FUNCTION_BLOCK FB_Test1000
VAR_INPUT
END_VAR
VAR_OUTPUT
END_VAR
VAR
	fbEvent: 			Tc3_Event.FB_Event;
	bVerbose:			BOOL;
	bInfo:				BOOL;
	bWarning:			BOOL;
	bError:				BOOL;
	bCritical:			BOOL;

END_VAR

fbEvent();

fbEvent.M_Error(832893823, 'Failed to ad recipe: %s %s');
fbEvent.M_Error(118851667, 'Gate interlock failed');
fbEvent.M_Error(697446562, 'Proximity sensor %s is faulty');
fbEvent.M_Error(810077404, 'System voltage is unstable');
fbEvent.M_Error(107227910, 'Data packet from robot is corrupt');
fbEvent.M_Error(478985983, 'Cylinder B did not retract within timeout');
fbEvent.M_Error(426179790, 'Main drive overtemperature');
fbEvent.M_Error(119981003, 'Network switch communication error');
fbEvent.M_Error(427933954, 'Operator login failed for user %s');
fbEvent.M_Error(373789771, 'Tool change failed on station %s');
fbEvent.M_Error(178323855, 'Regulator pressure is out of range');
fbEvent.M_Error(39012755, 'Homing failed for axis %s');
fbEvent.M_Error(980730346, 'Chiller fluid level is low');
fbEvent.M_Error(725753688, 'Vision system could not locate part %s');
fbEvent.M_Error(690645040, 'Fire suppression system activated');
fbEvent.M_Error(539036317, 'Motor B thermal overload');
fbEvent.M_Error(191893753, 'Analog input %s signal out of range');
fbEvent.M_Error(127546449, 'Palletizer stack height error');
fbEvent.M_Error(378168816, 'Failed to write to database');
fbEvent.M_Error(724256379, 'Inconsistent barcode scan for part %s');
fbEvent.M_Error(34792077, 'Axis %s software limit switch triggered');
fbEvent.M_Error(684752803, 'Manual mode interlock is active');
fbEvent.M_Error(65762173, 'Leak detected in hydraulic line %s');
fbEvent.M_Error(480483646, 'Pressure relief valve is active');
fbEvent.M_Error(839218, 'PLC CPU temperature is high');
fbEvent.M_Error(275778846, 'Cannot open file %s on HMI');
fbEvent.M_Error(254562129, 'Watchdog timer has expired');
fbEvent.M_Error(908391860, 'Clamping force not achieved');
fbEvent.M_Error(242273333, 'Emergency stop chain is broken');
fbEvent.M_Error(550219210, 'Proximity sensor 4 did not detect part');
fbEvent.M_Error(106098276, 'Axis 2 position deviation too high');
fbEvent.M_Error(309396701, 'Communication with VFD %s failed');
fbEvent.M_Error(922463265, 'Air filter is clogged');
fbEvent.M_Error(597666627, 'Incorrect part orientation detected');
fbEvent.M_Error(646335546, 'System failed to initialize');
fbEvent.M_Error(431554599, 'Torque limit exceeded for motor %s');
fbEvent.M_Error(569106138, 'Sensor supply voltage is low');
fbEvent.M_Error(263454198, 'Safety relay test failed');
fbEvent.M_Error(116099748, 'Cycle start not permitted: Guard open');
fbEvent.M_Error(121511879, 'Invalid command received from HMI');
fbEvent.M_Error(902925985, 'Conveyor speed is below setpoint');
fbEvent.M_Error(291757759, 'Failed to grip part at station %s');
fbEvent.M_Error(141691375, 'Hydraulic fluid level is critically low');
fbEvent.M_Error(790125858, 'Temperature sensor %s is disconnected');
fbEvent.M_Error(974334660, 'Robot is in singularity position');
fbEvent.M_Error(537205036, 'Network connection to SCADA lost');
fbEvent.M_Error(518848565, 'Axis %s hardware limit switch triggered');
fbEvent.M_Error(758816493, 'Pump motor failed to start');
fbEvent.M_Error(560430170, 'Mode change failed: System not in safe state');
fbEvent.M_Error(843353429, 'Error in motion group %s');
fbEvent.M_Error(54425602, 'Lubrication system fault');
fbEvent.M_Error(79236373, 'Failed to close valve %s');
fbEvent.M_Error(798717805, 'Excessive vibration detected on motor %s');
fbEvent.M_Error(416941017, 'Part presence sensor stuck on');
fbEvent.M_Error(833785224, 'Batch number %s is invalid or expired');
fbEvent.M_Error(884934701, 'Main circuit breaker is tripped');
fbEvent.M_Error(105321266, 'Failed to establish connection to robot %s');
fbEvent.M_Error(580072928, 'Pressure sensor reading is frozen');
fbEvent.M_Error(478251424, 'Cylinder A extended unexpectedly');
fbEvent.M_Error(715796097, 'Insufficient air pressure for gripper');
fbEvent.M_Error(916964646, 'E-Stop reset failed: Fault condition still present');
fbEvent.M_Error(352575033, 'Encoder battery voltage is low');
fbEvent.M_Error(845967336, 'Invalid parameter set for drive %s');
fbEvent.M_Error(400399278, 'Flow rate is too low in line %s');
fbEvent.M_Error(594607632, 'Homing sequence interrupted');
fbEvent.M_Error(576534155, 'Safety mat is active');
fbEvent.M_Error(101312224, 'PLC scan time is too high');
fbEvent.M_Error(630778805, 'Configuration file %s is corrupted');
fbEvent.M_Error(11187824, 'Axis %s stalled during movement');
fbEvent.M_Error(406567956, 'Temperature out of spec for oven %s');
fbEvent.M_Error(122069157, 'Failed to eject part from mold');
fbEvent.M_Error(653459603, 'Wrong tool loaded in spindle');
fbEvent.M_Error(315127736, 'Robot path planning error for destination %s');
fbEvent.M_Error(532962581, 'Overvoltage detected on DC bus');
fbEvent.M_Error(990252450, 'Purge cycle failed to complete');
fbEvent.M_Error(80896362, 'Signal conflict between two sensors');
fbEvent.M_Error(956082325, 'Cannot load G-code file: %s');
fbEvent.M_Error(716456626, 'Failed to enable drive group %s');
fbEvent.M_Error(954893308, 'Reservoir level is high');
fbEvent.M_Error(785582455, 'Welding tip is worn');
fbEvent.M_Error(103430303, 'Incorrect fixture ID %s received');
fbEvent.M_Error(707539160, 'Servo motor overheating');
fbEvent.M_Error(515304940, 'Failed to close safety gate');
fbEvent.M_Error(28063579, 'Sensor fault: Short circuit');
fbEvent.M_Error(619031287, 'PLC memory is full');
fbEvent.M_Error(894005669, 'Actuator %s did not complete motion');
fbEvent.M_Error(323445774, 'Part quality check failed at station %s');
fbEvent.M_Error(366731016, 'Main contactor did not engage');
fbEvent.M_Error(194019962, 'System is in E-Stop state');
fbEvent.M_Error(932272750, 'Analog output %s is at fault');
fbEvent.M_Error(6921616, 'Failed to read data from RFID tag');
fbEvent.M_Error(528281057, 'Conveyor index timeout');
fbEvent.M_Error(738673258, 'Emergency stop line is broken');
fbEvent.M_Error(108292847, 'Axis %s is not referenced');
fbEvent.M_Error(10066866, 'Valve manifold communication error');
fbEvent.M_Error(436001307, 'Temperature ramp rate too fast');
fbEvent.M_Error(281793927, 'Failed to synchronize axes');
fbEvent.M_Error(547426220, 'Robot joint %s limit exceeded');
fbEvent.M_Error(250102496, 'Vision system lighting failure');
fbEvent.M_Error(680495858, 'Pressure sensor %s shows maximum value');
fbEvent.M_Error(882166272, 'Machine not homed');
fbEvent.M_Error(532755668, 'User %s does not have required permissions');
fbEvent.M_Error(246357126, 'Hydraulic accumulator is pre-charged incorrectly');
fbEvent.M_Error(132892386, 'Coolant flow switch is open');
fbEvent.M_Error(286233919, 'Part jam detected in chute %s');
fbEvent.M_Error(598877655, 'Failed to zero axis %s');
fbEvent.M_Error(790152895, 'Motor phase loss detected');
fbEvent.M_Error(707430004, 'Internal PLC error: Task overrun');
fbEvent.M_Error(848312986, 'Barcode scanner not ready');
fbEvent.M_Error(122916115, 'Invalid move command for axis %s');
fbEvent.M_Error(741153201, 'Safety PLC communication fault');
fbEvent.M_Error(879449371, 'Filter differential pressure is high');
fbEvent.M_Error(28238082, 'Cylinder B pressure not building');
fbEvent.M_Error(894279110, 'Spindle speed not reached');
fbEvent.M_Error(500211574, 'Robot collision detected');
fbEvent.M_Error(433875535, 'Failed to update recipe %s in database');
fbEvent.M_Error(675711322, 'Interlock condition not met for operation %s');
fbEvent.M_Error(816986360, 'System pressure is too high');
fbEvent.M_Error(843994824, 'VFD in fault state');
fbEvent.M_Error(282577562, 'HMI backup failed');
fbEvent.M_Error(654845819, 'Position feedback lost for axis %s');
fbEvent.M_Error(755383388, 'Label printer error: Out of labels');
fbEvent.M_Error(840940439, 'Chiller temperature is too high');
fbEvent.M_Error(726897854, 'Part unloading failed');
fbEvent.M_Error(544112161, 'Emergency stop reset timeout');
fbEvent.M_Error(738601621, 'Axis %s command position and actual position mismatch');
fbEvent.M_Error(947294229, 'Pump is running dry');
fbEvent.M_Error(487525630, 'Level sensor in tank %s is faulted');
fbEvent.M_Error(277091341, 'Failed to park robot');
fbEvent.M_Error(792913450, 'Conveyor motor overload');
fbEvent.M_Error(198407162, 'Wrong material loaded for job %s');
fbEvent.M_Error(477836306, 'Air compressor fault');
fbEvent.M_Error(709412327, 'PLC I/O module error');
fbEvent.M_Error(262982191, 'Excessive cycle time detected');
fbEvent.M_Error(458184506, 'Safety gate switch is welded');
fbEvent.M_Error(456148294, 'Failed to open valve %s');
fbEvent.M_Error(179389617, 'Thermocouple %s is broken');
fbEvent.M_Error(373226799, 'Cylinder A failed to extend');
fbEvent.M_Error(217544684, 'Robot is not in auto mode');
fbEvent.M_Error(289058555, 'System failed to shutdown gracefully');
fbEvent.M_Error(881340240, 'Load cell signal is unstable');
fbEvent.M_Error(426479410, 'Homing timeout for axis %s');
fbEvent.M_Error(368079717, 'Purge valve is stuck open');
fbEvent.M_Error(901417390, 'Network cable unplugged for device %s');
fbEvent.M_Error(119729734, 'Operator intervention required');
fbEvent.M_Error(817664351, 'Failed to apply torque on fastener %s');
fbEvent.M_Error(348454004, 'Proximity sensor fault: Wire break');
fbEvent.M_Error(103013536, 'Main power supply failure');
fbEvent.M_Error(17242893, 'Robot program %s is not found');
fbEvent.M_Error(530604795, 'VFD overcurrent trip');
fbEvent.M_Error(563485368, 'Cylinder B failed to retract');
fbEvent.M_Error(170043574, 'Failed to maintain pressure at %s bar');
fbEvent.M_Error(329133, 'Axis %s brake did not release');
fbEvent.M_Error(844021694, 'HMI screen saver is active');
fbEvent.M_Error(578481480, 'Failed to enable safety outputs');
fbEvent.M_Error(499147908, 'Part transfer failed');
fbEvent.M_Error(815311898, 'Incorrect password entered %s times');
fbEvent.M_Error(386296766, 'Sensor %s is dirty or misaligned');
fbEvent.M_Error(157727822, 'Spindle tool not clamped');
fbEvent.M_Error(865519035, 'System is in maintenance mode');
fbEvent.M_Error(336598871, 'Failed to log data to file %s');
fbEvent.M_Error(635260245, 'Conveyor belt slipped');
fbEvent.M_Error(776980042, 'Hydraulic fluid is contaminated');
fbEvent.M_Error(949104028, 'Robot joint %s temperature is high');
fbEvent.M_Error(592920496, 'Axis 3 move command cancelled');
fbEvent.M_Error(54844710, 'Light curtain fault: Mutingshort circuit');
fbEvent.M_Error(869858701, 'PLC battery needs replacement');
fbEvent.M_Error(718470536, 'Failed to connect to MES system');
fbEvent.M_Error(684582860, 'Weight of part %s is out of tolerance');
fbEvent.M_Error(802205547, 'Air dryer fault');
fbEvent.M_Error(621187246, 'Valve %s did not shift');
fbEvent.M_Error(418538085, 'Safety relay did not pick up');
fbEvent.M_Error(951020145, 'Failed to find reference mark for axis %s');
fbEvent.M_Error(6730302, 'Temperature in zone %s is too low');
fbEvent.M_Error(976382904, 'Clamp pressure not released');
fbEvent.M_Error(818586704, 'Robot path obstructed');
fbEvent.M_Error(479810162, 'Failed to save settings to HMI');
fbEvent.M_Error(423729794, 'Motor B is not responding');
fbEvent.M_Error(417051589, 'Proximity sensor %s is always on');
fbEvent.M_Error(619244592, 'System pressure not building');
fbEvent.M_Error(909197747, 'Failed to execute command %s');
fbEvent.M_Error(973694476, 'E-Stop source: Panel Button');
fbEvent.M_Error(159508959, 'Axis %s is disabled');
fbEvent.M_Error(638220346, 'Pump suction is clogged');
fbEvent.M_Error(201076670, 'Failed to read configuration from drive');
fbEvent.M_Error(357632549, 'Part height is incorrect at station %s');
fbEvent.M_Error(357999834, 'Robot is in singularity, cannot move');
fbEvent.M_Error(596581822, 'VFD undervoltage fault');
fbEvent.M_Error(902198983, 'Cylinder A pressure sensor fault');
fbEvent.M_Error(925673804, 'Safety gate not locked');
fbEvent.M_Error(730111847, 'Failed to write to I/O module %s');
fbEvent.M_Error(187095213, 'Encoder resolution mismatch');
fbEvent.M_Error(165625991, 'Spindle speed is zero');
fbEvent.M_Error(437415664, 'System failed to enter run mode');
fbEvent.M_Error(635973644, 'Pallet not present at location %s');
fbEvent.M_Error(370392395, 'Hydraulic return filter is clogged');
fbEvent.M_Error(7449781, 'Robot gripper failed to open');
fbEvent.M_Error(348878313, 'PLC time sync failed');
fbEvent.M_Error(990092022, 'Failed to find part %s in vision system');
fbEvent.M_Error(458919012, 'Conveyor tracking lost');
fbEvent.M_Error(770244041, 'Emergency stop source: Pull Cord');
fbEvent.M_Error(185356685, 'Axis %s brake did not engage');
fbEvent.M_Error(449988299, 'Motor A thermal model trip');
fbEvent.M_Error(835758112, 'Level sensor in tank %s is frozen');
fbEvent.M_Error(811924027, 'Failed to close gripper');
fbEvent.M_Error(64576557, 'Safety light curtain is muted');
fbEvent.M_Error(967372774, 'VFD DC bus overvoltage');
fbEvent.M_Error(216876843, 'Cylinder B extended unexpectedly');
fbEvent.M_Error(668341244, 'Failed to start cycle: Guard not closed');
fbEvent.M_Error(839807760, 'Robot is in manual mode');
fbEvent.M_Error(109044549, 'System pressure relief valve active');
fbEvent.M_Error(963090393, 'Failed to load G-code: Invalid syntax');
fbEvent.M_Error(88367024, 'Axis %s is not homed');
fbEvent.M_Error(305668940, 'Motor C bearing failure');
fbEvent.M_Error(80432916, 'Air pressure is too high');
fbEvent.M_Error(360463664, 'Failed to park robot in home position');
fbEvent.M_Error(973132419, 'HMI firmware update failed');
fbEvent.M_Error(757446510, 'E-Stop source: Gateway');
fbEvent.M_Error(584607011, 'Proximity sensor %s is always off');
fbEvent.M_Error(560041746, 'Temperature ramp rate too slow');
fbEvent.M_Error(773247963, 'Failed to open gripper');
fbEvent.M_Error(85107326, 'Robot collision detected at joint %s');
fbEvent.M_Error(237489277, 'VFD motor stall');
fbEvent.M_Error(824859949, 'Cylinder A failed to retract');
fbEvent.M_Error(61467370, 'Failed to maintain speed at %s RPM');
fbEvent.M_Error(2628015, 'Safety PLC test failed');
fbEvent.M_Error(186098607, 'Failed to read barcode from part %s');
fbEvent.M_Error(417246690, 'Conveyor motor is not running');
fbEvent.M_Error(691255652, 'Emergency stop source: Safety Mat');
fbEvent.M_Error(635356995, 'Axis %s is in alarm state');
fbEvent.M_Error(265437496, 'Pump discharge is blocked');
fbEvent.M_Error(958296709, 'Failed to execute robot program %s');
fbEvent.M_Error(405885388, 'System is in E-Stop state: Reset required');
fbEvent.M_Error(50258952, 'Motor D overtemperature');
fbEvent.M_Error(103822728, 'Air leak detected in circuit %s');
fbEvent.M_Error(585336403, 'Failed to close valve manifold');
fbEvent.M_Error(133950658, 'Safety gate not closed');
fbEvent.M_Error(350665306, 'Failed to set output %s');
fbEvent.M_Error(614113915, 'Encoder count error');
fbEvent.M_Error(996015977, 'Spindle direction is incorrect');
fbEvent.M_Error(329884446, 'System failed to initialize I/O');
fbEvent.M_Error(381300644, 'Pallet is skewed at location %s');
fbEvent.M_Error(894443599, 'Hydraulic pump is noisy');
fbEvent.M_Error(564280028, 'Robot gripper failed to close');
fbEvent.M_Error(138989844, 'PLC network redundancy lost');
fbEvent.M_Error(798245427, 'Failed to find fiducial %s in vision system');
fbEvent.M_Error(873836778, 'Conveyor belt is torn');
fbEvent.M_Error(36049922, 'Emergency stop source: Dual Channel');
fbEvent.M_Error(788139320, 'Axis %s following error is active');
fbEvent.M_Error(240236294, 'Motor E bearing temperature is high');
fbEvent.M_Error(542290731, 'Air pressure is too low');
fbEvent.M_Error(408567347, 'Failed to move robot to safe position');
fbEvent.M_Error(878151236, 'HMI application crashed');
fbEvent.M_Error(753128079, 'E-Stop source: Hardwired');
fbEvent.M_Error(227807103, 'Proximity sensor %s is intermittent');
fbEvent.M_Error(463877781, 'Temperature overshoot detected');
fbEvent.M_Error(277757321, 'Failed to release part');
fbEvent.M_Error(182345328, 'Robot joint limit reached');
fbEvent.M_Error(302203944, 'VFD motor overload');
fbEvent.M_Error(478251424, 'Cylinder A extended unexpectedly');
fbEvent.M_Error(802928548, 'Failed to maintain torque at %s Nm');
fbEvent.M_Error(887612404, 'Safety relay test passed with warnings');
fbEvent.M_Error(212140868, 'Failed to write barcode to part %s');
fbEvent.M_Error(379744884, 'Conveyor speed is zero');
fbEvent.M_Error(170151812, 'Emergency stop source: Unlisted');
fbEvent.M_Error(885967005, 'Axis %s is not enabled');
fbEvent.M_Error(396387794, 'Pump cavitation detected');
fbEvent.M_Error(404055868, 'Failed to load robot program %s');
fbEvent.M_Error(406348215, 'System is in fault state: Reset required');
fbEvent.M_Error(919838823, 'Motor F overcurrent');
fbEvent.M_Error(233061244, 'Air dryer is saturated');
fbEvent.M_Error(186408788, 'Failed to open safety valve');
fbEvent.M_Error(913386085, 'Safety gate is not interlocked');
fbEvent.M_Error(741030180, 'Failed to clear output %s');
fbEvent.M_Error(583691718, 'Encoder signal is noisy');
fbEvent.M_Error(450171867, 'Spindle tool is broken');
fbEvent.M_Error(90116955, 'System failed to load configuration');
fbEvent.M_Error(155930849, 'Pallet is missing at location %s');
fbEvent.M_Error(966835846, 'Hydraulic fluid is low');
fbEvent.M_Error(564997759, 'Robot gripper is worn');
fbEvent.M_Error(791956772, 'PLC task watchdog has expired');
fbEvent.M_Error(829423237, 'Failed to match pattern %s in vision system');
fbEvent.M_Error(666584115, 'Conveyor motor is overheating');
fbEvent.M_Error(996676608, 'Emergency stop source: Software');
fbEvent.M_Error(991067110, 'Axis %s is in warning state');
fbEvent.M_Error(30615213, 'Motor G is not calibrated');
fbEvent.M_Error(57826245, 'Air pressure is unstable');
fbEvent.M_Error(286572655, 'Failed to power down robot');
fbEvent.M_Error(440680958, 'HMI display is faulty');
fbEvent.M_Error(692138795, 'E-Stop source: External');
fbEvent.M_Error(676144596, 'Proximity sensor %s is miswired');
fbEvent.M_Error(75459534, 'Temperature undershoot detected');
fbEvent.M_Error(194196433, 'Failed to grip part');
fbEvent.M_Error(528206401, 'Robot software limit reached');
fbEvent.M_Error(489457463, 'VFD communication is lost');
fbEvent.M_Error(111852218, 'Cylinder B failed to extend');
fbEvent.M_Error(103224179, 'Failed to maintain position at %s mm');
fbEvent.M_Error(539163415, 'Safety relay test failed critically');
fbEvent.M_Error(677923405, 'Failed to verify barcode on part %s');
fbEvent.M_Error(973083953, 'Conveyor is overloaded');
fbEvent.M_Error(400783557, 'Emergency stop source: Unknown');
fbEvent.M_Error(621913516, 'Axis %s is in fault state');
fbEvent.M_Error(350444340, 'Pump efficiency is low');
fbEvent.M_Error(634344537, 'Failed to save robot program %s');
fbEvent.M_Error(174850429, 'System is in safe state');
fbEvent.M_Error(136101471, 'Motor H has a ground fault');
fbEvent.M_Error(300947899, 'Air filter is dirty');
fbEvent.M_Error(449292690, 'Failed to close isolation valve');
fbEvent.M_Error(424789367, 'Safety gate is open');
fbEvent.M_Error(409216181, 'Failed to set input %s');
fbEvent.M_Error(933027441, 'Encoder battery is dead');
fbEvent.M_Error(651826221, 'Spindle is not running');
fbEvent.M_Error(731123442, 'System failed to boot');
fbEvent.M_Error(939430834, 'Pallet is double-stacked at location %s');
fbEvent.M_Error(198827357, 'Hydraulic fluid is overheating');
fbEvent.M_Error(751844004, 'Robot gripper is damaged');
fbEvent.M_Error(311451049, 'PLC scan time is too long');
fbEvent.M_Error(660322600, 'Failed to locate feature %s in vision system');
fbEvent.M_Error(476336752, 'Conveyor belt is misaligned');
fbEvent.M_Error(309335721, 'Emergency stop has been reset');
fbEvent.M_Error(634474780, 'Axis %s is homed');
fbEvent.M_Error(663037999, 'Motor I is not configured');
fbEvent.M_Error(142099094, 'Air pressure is normal');
fbEvent.M_Error(472951340, 'Failed to power on robot');
fbEvent.M_Error(564592578, 'HMI is connected');
fbEvent.M_Error(293993190, 'E-Stop source is clear');
fbEvent.M_Error(944357119, 'Proximity sensor %s is working');
fbEvent.M_Error(530241786, 'Temperature is stable');
fbEvent.M_Error(321847964, 'Part is gripped');
fbEvent.M_Error(687503128, 'Robot is in home position');
fbEvent.M_Error(755155798, 'VFD is running');
fbEvent.M_Error(765643058, 'Cylinder A is retracted');
fbEvent.M_Error(726804838, 'Position is correct at %s mm');
fbEvent.M_Error(796973120, 'Safety system is OK');
fbEvent.M_Error(603145075, 'Barcode on part %s is verified');
fbEvent.M_Error(397074462, 'Conveyor is running');
fbEvent.M_Error(154609732, 'System is in run mode');
fbEvent.M_Error(49686060, 'Axis %s is enabled');
fbEvent.M_Error(943047633, 'Pump is running');
fbEvent.M_Error(457848118, 'Robot program %s is loaded');
fbEvent.M_Error(732406110, 'System is ready');
fbEvent.M_Error(524031458, 'Motor J is OK');
fbEvent.M_Error(175987386, 'Air system is OK');
fbEvent.M_Error(453988495, 'Valve is open');
fbEvent.M_Error(540011896, 'Safety gate is closed and locked');
fbEvent.M_Error(279662546, 'Input %s is on');
fbEvent.M_Error(529208917, 'Encoder is working');
fbEvent.M_Error(956407335, 'Spindle is at speed');
fbEvent.M_Error(995454603, 'System is booted');
fbEvent.M_Error(181892822, 'Pallet is at location %s');
fbEvent.M_Error(283109924, 'Hydraulic system is OK');
fbEvent.M_Error(525919964, 'Robot gripper is open');
fbEvent.M_Error(755154645, 'PLC is running');
fbEvent.M_Error(984938963, 'Vision system is ready');
fbEvent.M_Error(827863662, 'Conveyor is stopped');
fbEvent.M_Error(702570581, 'System is in auto mode');
fbEvent.M_Error(614863977, 'Axis %s is stopped');
fbEvent.M_Error(526801336, 'Pump is stopped');
fbEvent.M_Error(6496515, 'Robot is idle');
fbEvent.M_Error(569656297, 'System is in manual mode');
fbEvent.M_Error(792582087, 'Motor K is stopped');
fbEvent.M_Error(353171688, 'Air system is off');
fbEvent.M_Error(548874609, 'Valve is closed');
fbEvent.M_Error(693263043, 'Safety gate is unlocked');
fbEvent.M_Error(264507605, 'Input %s is off');
fbEvent.M_Error(533849785, 'Encoder is not connected');
fbEvent.M_Error(745304882, 'Spindle is stopped');
fbEvent.M_Error(542239548, 'System is shutting down');
fbEvent.M_Error(87711744, 'Pallet is empty at location %s');
fbEvent.M_Error(93283491, 'Hydraulic system is off');
fbEvent.M_Error(361966966, 'Robot gripper is closed');
fbEvent.M_Error(635796636, 'PLC is stopped');
fbEvent.M_Error(941407936, 'Vision system is off');
fbEvent.M_Error(373346217, 'Conveyor is jammed');
fbEvent.M_Error(770631599, 'System is in fault');
fbEvent.M_Error(971819022, 'Axis %s is moving');
fbEvent.M_Error(944421970, 'Pump is priming');
fbEvent.M_Error(259892226, 'Robot is moving');
fbEvent.M_Error(181859858, 'System is initializing');
fbEvent.M_Error(276810072, 'Motor L is starting');
fbEvent.M_Error(90775392, 'Air system is charging');
fbEvent.M_Error(172701248, 'Valve is shifting');
fbEvent.M_Error(961944472, 'Safety gate is opening');
fbEvent.M_Error(418224237, 'Input %s is faulted');
fbEvent.M_Error(455563805, 'Encoder is homing');
fbEvent.M_Error(663806485, 'Spindle is starting');
fbEvent.M_Error(761487350, 'System is saving data');
fbEvent.M_Error(206145070, 'Pallet is arriving at location %s');
fbEvent.M_Error(881436336, 'Hydraulic system is charging');
fbEvent.M_Error(617228608, 'Robot gripper is releasing');
fbEvent.M_Error(207776615, 'PLC is in program mode');
fbEvent.M_Error(807848533, 'Vision system is capturing image');
fbEvent.M_Error(41725285, 'Conveyor is indexing');
fbEvent.M_Error(57280963, 'System is in config mode');
fbEvent.M_Error(544086596, 'Axis %s is referencing');
fbEvent.M_Error(335007187, 'Pump is building pressure');
fbEvent.M_Error(361844212, 'Robot is referencing');
fbEvent.M_Error(338315346, 'System is in test mode');
fbEvent.M_Error(47527036, 'Motor M is running');
fbEvent.M_Error(833767271, 'Air system is at pressure');
fbEvent.M_Error(95999827, 'Valve is energized');
fbEvent.M_Error(700847574, 'Safety gate is closing');
fbEvent.M_Error(849363082, 'Input %s is simulated');
fbEvent.M_Error(340828109, 'Encoder is synchronized');
fbEvent.M_Error(407073985, 'Spindle is braking');
fbEvent.M_Error(813120861, 'System is online');
fbEvent.M_Error(861139381, 'Pallet is leaving location %s');
fbEvent.M_Error(365218255, 'Hydraulic system is active');
fbEvent.M_Error(618186036, 'Robot gripper is gripping');
fbEvent.M_Error(915053279, 'PLC is in run mode');
fbEvent.M_Error(826798443, 'Vision system is processing image');
fbEvent.M_Error(360021832, 'Conveyor is accelerating');
fbEvent.M_Error(109320720, 'System is in service mode');
fbEvent.M_Error(712668444, 'Axis %s is waiting');
fbEvent.M_Error(140194638, 'Pump is at speed');
fbEvent.M_Error(413280508, 'Robot is waiting for input');
fbEvent.M_Error(305123578, 'System is in standby');
fbEvent.M_Error(577509354, 'Motor N is at temperature');
fbEvent.M_Error(322923140, 'Air system is venting');
fbEvent.M_Error(125674975, 'Valve is de-energized');
fbEvent.M_Error(305819171, 'Safety gate is locked');
fbEvent.M_Error(401867310, 'Input %s is forced');
fbEvent.M_Error(262738951, 'Encoder is at zero');
fbEvent.M_Error(105901330, 'Spindle is changing tool');
fbEvent.M_Error(217052528, 'System is offline');
fbEvent.M_Error(844887995, 'Pallet is at position %s');
fbEvent.M_Error(608989523, 'Hydraulic system is idle');
fbEvent.M_Error(717765502, 'Robot gripper is empty');
fbEvent.M_Error(240773138, 'PLC is in fault mode');
fbEvent.M_Error(911204631, 'Vision system failed to focus');
fbEvent.M_Error(57039477, 'Conveyor is decelerating');
fbEvent.M_Error(163495912, 'System is in emergency stop');
fbEvent.M_Error(16864990, 'Axis %s is in error');
fbEvent.M_Error(377623810, 'Pump is in alarm');
fbEvent.M_Error(779282330, 'Robot is in error');
fbEvent.M_Error(258163367, 'System is in safe stop');
fbEvent.M_Error(766331159, 'Motor O is in alarm');
fbEvent.M_Error(736968920, 'Air system is in fault');
fbEvent.M_Error(925602966, 'Valve is in fault');
fbEvent.M_Error(645750778, 'Safety gate is in fault');
fbEvent.M_Error(626477413, 'Input %s is in error');
fbEvent.M_Error(325226080, 'Encoder is in alarm');
fbEvent.M_Error(442704929, 'Spindle is in fault');
fbEvent.M_Error(454848228, 'System is in power save');
fbEvent.M_Error(339227309, 'Pallet is damaged at location %s');
fbEvent.M_Error(74315214, 'Hydraulic system is in fault');
fbEvent.M_Error(22088896, 'Robot gripper is in fault');
fbEvent.M_Error(572326510, 'PLC is in stop mode');
fbEvent.M_Error(516754421, 'Vision system is in error');
fbEvent.M_Error(340190816, 'Conveyor is in E-Stop');
fbEvent.M_Error(579673878, 'System is in maintenance');
fbEvent.M_Error(159508959, 'Axis %s is disabled');
fbEvent.M_Error(964219551, 'Pump is disabled');
fbEvent.M_Error(683696240, 'Robot is disabled');
fbEvent.M_Error(557066724, 'System is in setup');
fbEvent.M_Error(165858997, 'Motor P is disabled');
fbEvent.M_Error(234731108, 'Air system is disabled');
fbEvent.M_Error(655951572, 'Valve is disabled');
fbEvent.M_Error(62951896, 'Safety gate is disabled');
fbEvent.M_Error(904304221, 'Input %s is disabled');
fbEvent.M_Error(159027536, 'Encoder is disabled');
fbEvent.M_Error(289949864, 'Spindle is disabled');
fbEvent.M_Error(319110611, 'System is in reset');
fbEvent.M_Error(667308375, 'Pallet is missing from location %s');
fbEvent.M_Error(824981369, 'Hydraulic system is disabled');
fbEvent.M_Error(170426620, 'Robot gripper is disabled');
fbEvent.M_Error(108431048, 'PLC is in reset');
fbEvent.M_Error(570763187, 'Vision system is disabled');
fbEvent.M_Error(499438490, 'Conveyor is in reset');
fbEvent.M_Error(526591558, 'System is in power up');
fbEvent.M_Error(111094027, 'Axis %s is powering up');
fbEvent.M_Error(110725211, 'Pump is powering up');
fbEvent.M_Error(104405939, 'Robot is powering up');
fbEvent.M_Error(866629375, 'System is in power down');
fbEvent.M_Error(264569568, 'Motor Q is powering down');
fbEvent.M_Error(482613552, 'Air system is powering down');
fbEvent.M_Error(58824455, 'Valve is powering down');
fbEvent.M_Error(234602243, 'Safety gate is powering down');
fbEvent.M_Error(624719034, 'Input %s is powering down');
fbEvent.M_Error(692011725, 'Encoder is powering down');
fbEvent.M_Error(822934053, 'Spindle is powering down');
fbEvent.M_Error(307361688, 'System is in communication fault');
fbEvent.M_Error(327357878, 'Pallet is wrong at location %s');
fbEvent.M_Error(221046379, 'Hydraulic system is in communication fault');
fbEvent.M_Error(365980608, 'Robot gripper is in communication fault');
fbEvent.M_Error(90860287, 'PLC is in communication fault');
fbEvent.M_Error(766317175, 'Vision system is in communication fault');
fbEvent.M_Error(415163047, 'Conveyor is in communication fault');
fbEvent.M_Error(149896403, 'System is in configuration fault');
fbEvent.M_Error(345061979, 'Axis %s is in configuration fault');
fbEvent.M_Error(130294318, 'Pump is in configuration fault');
fbEvent.M_Error(828462898, 'Robot is in configuration fault');
fbEvent.M_Error(230789099, 'System is in hardware fault');
fbEvent.M_Error(475894515, 'Motor R is in hardware fault');
fbEvent.M_Error(986432188, 'Air system is in hardware fault');
fbEvent.M_Error(694796410, 'Valve is in hardware fault');
fbEvent.M_Error(875891613, 'Safety gate is in hardware fault');
fbEvent.M_Error(511865723, 'Input %s is in hardware fault');
fbEvent.M_Error(337610281, 'Encoder is in hardware fault');
fbEvent.M_Error(681484970, 'Lag error');
fbEvent.M_Error(774527956, 'Lag error 2');
fbEvent.M_Error(103668540, 'Lag error 3');

PROPERTY PUBLIC P_Event : reference to FB_event
GET
P_Event ref= fbEvent;
END_GET
END_PROPERTY

END_FUNCTION_BLOCK

(* stored: Version 1.1.0.1
   POU FB_Test1000: Id {10fc8182-56aa-4c15-8394-db1fa4a2f8e5}, SpecialFunc None
   Property P_Event: Id {c9963adf-3970-4f81-9f65-c4cce93fef12}
   Get Get: Id {164e6f1a-62a7-4f2e-8ee2-e70cbc651471} *)
